PROGRAM Stn10
VAR

	start10: BOOL;
	reset10: BOOL;

	Stn10ProcessFE: F_TRIG;
	Stn10ProcessRE: R_TRIG;
	bCutStn10ProcessHalt: BOOL;
	DoorClose10: R_TRIG;
	bStn10DoorClamp: BOOL;

END_VAR
VAR // added by the converter: edge detectors and wires of the graphical bodies
    _w1, _w2 : ANY;
END_VAR

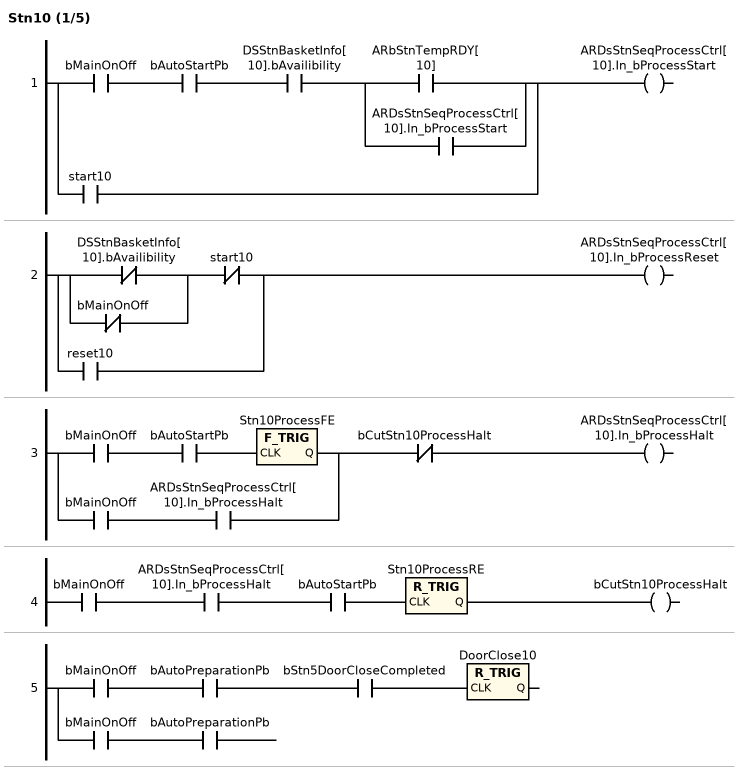
// NETWORK 1
ARDsStnSeqProcessCtrl[10].In_bProcessStart := bMainOnOff AND bAutoStartPb AND DSStnBasketInfo[10].bAvailibility AND (ARbStnTempRDY[10] OR ARDsStnSeqProcessCtrl[10].In_bProcessStart) OR start10;

// NETWORK 2
ARDsStnSeqProcessCtrl[10].In_bProcessReset := (NOT DSStnBasketInfo[10].bAvailibility OR NOT bMainOnOff) AND NOT start10 OR reset10;

// NETWORK 3
Stn10ProcessFE(CLK := bMainOnOff AND bAutoStartPb); // F_TRIG
ARDsStnSeqProcessCtrl[10].In_bProcessHalt := (Stn10ProcessFE.Q OR bMainOnOff AND ARDsStnSeqProcessCtrl[10].In_bProcessHalt) AND NOT bCutStn10ProcessHalt;

// NETWORK 4
Stn10ProcessRE(CLK := bMainOnOff AND ARDsStnSeqProcessCtrl[10].In_bProcessHalt AND bAutoStartPb); // R_TRIG
bCutStn10ProcessHalt := Stn10ProcessRE.Q;

// NETWORK 5
DoorClose10(CLK := bMainOnOff AND bAutoPreparationPb AND bStn5DoorCloseCompleted); // R_TRIG
(* DoorClose10.Q OR bMainOnOff AND bAutoPreparationPb; result not used *)

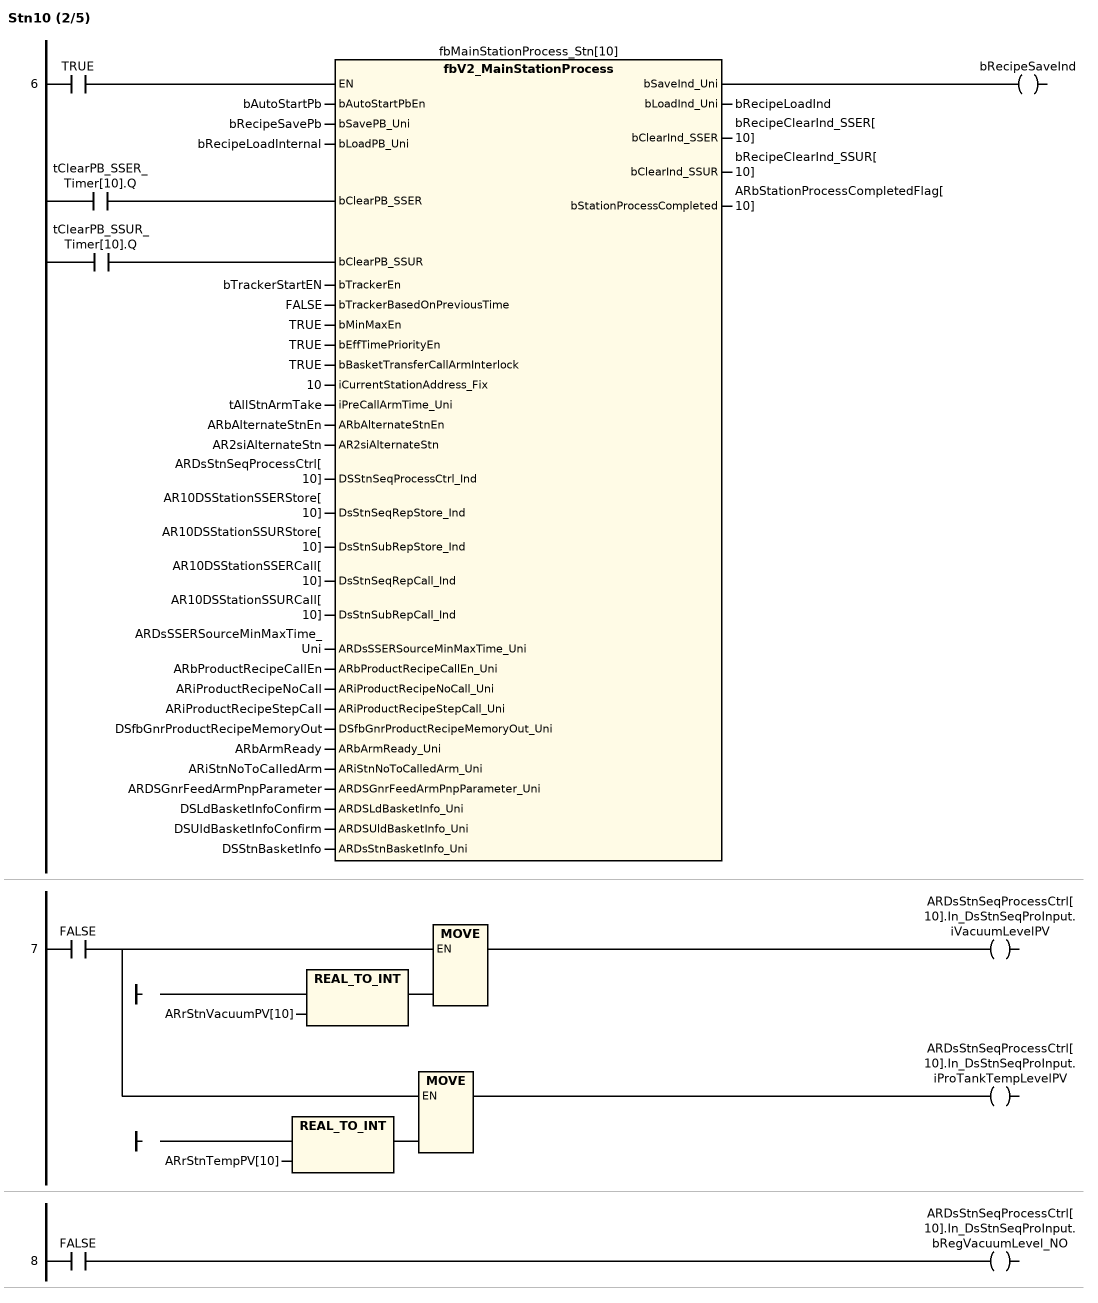
// NETWORK 6
fbMainStationProcess_Stn[10](
    bAutoStartPbEn := bAutoStartPb,
    bSavePB_Uni := bRecipeSavePb,
    bLoadPB_Uni := bRecipeLoadInternal,
    bClearPB_SSER := tClearPB_SSER_Timer[10].Q,
    bClearPB_SSUR := tClearPB_SSUR_Timer[10].Q,
    bTrackerEn := bTrackerStartEN,
    bTrackerBasedOnPreviousTime := FALSE,
    bMinMaxEn := TRUE,
    bEffTimePriorityEn := TRUE,
    bBasketTransferCallArmInterlock := TRUE,
    iCurrentStationAddress_Fix := 10,
    iPreCallArmTime_Uni := tAllStnArmTake,
    ARbAlternateStnEn := ARbAlternateStnEn,
    AR2siAlternateStn := AR2siAlternateStn,
    DSStnSeqProcessCtrl_Ind := ARDsStnSeqProcessCtrl[10],
    DsStnSeqRepStore_Ind := AR10DSStationSSERStore[10],
    DsStnSubRepStore_Ind := AR10DSStationSSURStore[10],
    DsStnSeqRepCall_Ind := AR10DSStationSSERCall[10],
    DsStnSubRepCall_Ind := AR10DSStationSSURCall[10],
    ARDsSSERSourceMinMaxTime_Uni := ARDsSSERSourceMinMaxTime_Uni,
    ARbProductRecipeCallEn_Uni := ARbProductRecipeCallEn,
    ARiProductRecipeNoCall_Uni := ARiProductRecipeNoCall,
    ARiProductRecipeStepCall_Uni := ARiProductRecipeStepCall,
    DSfbGnrProductRecipeMemoryOut_Uni := DSfbGnrProductRecipeMemoryOut,
    ARbArmReady_Uni := ARbArmReady,
    ARiStnNoToCalledArm_Uni := ARiStnNoToCalledArm,
    ARDSGnrFeedArmPnpParameter_Uni := ARDSGnrFeedArmPnpParameter,
    ARDSLdBasketInfo_Uni := DSLdBasketInfoConfirm,
    ARDSUldBasketInfo_Uni := DSUldBasketInfoConfirm,
    ARDsStnBasketInfo_Uni := DSStnBasketInfo,
    bLoadInd_Uni => bRecipeLoadInd,
    bClearInd_SSER => bRecipeClearInd_SSER[10],
    bClearInd_SSUR => bRecipeClearInd_SSUR[10],
    bStationProcessCompleted => ARbStationProcessCompletedFlag[10]); // fbV2_MainStationProcess
bRecipeSaveInd := fbMainStationProcess_Stn[10].bSaveInd_Uni;

// NETWORK 7
IF FALSE THEN _w1 := REAL_TO_INT(ARrStnVacuumPV[10]); END_IF
ARDsStnSeqProcessCtrl[10].In_DsStnSeqProInput.iVacuumLevelPV := _w1;
IF FALSE THEN _w2 := REAL_TO_INT(ARrStnTempPV[10]); END_IF
ARDsStnSeqProcessCtrl[10].In_DsStnSeqProInput.iProTankTempLevelPV := _w2;

// NETWORK 8
ARDsStnSeqProcessCtrl[10].In_DsStnSeqProInput.bRegVacuumLevel_NO := FALSE;

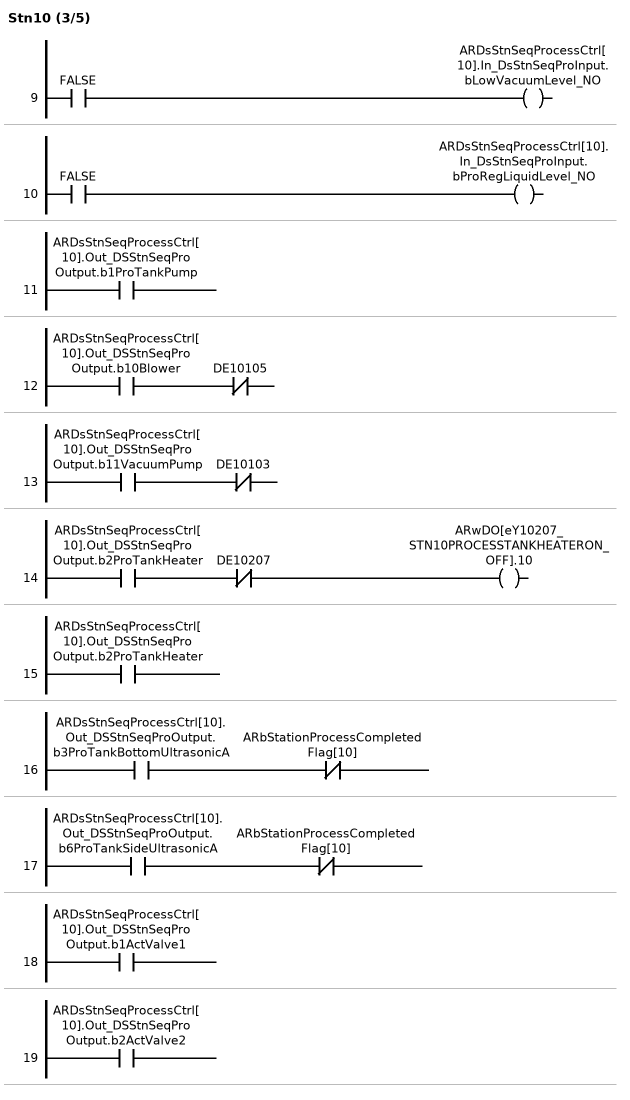
// NETWORK 9
ARDsStnSeqProcessCtrl[10].In_DsStnSeqProInput.bLowVacuumLevel_NO := FALSE;

// NETWORK 10
ARDsStnSeqProcessCtrl[10].In_DsStnSeqProInput.bProRegLiquidLevel_NO := FALSE;

// NETWORK 11
(* ARDsStnSeqProcessCtrl[10].Out_DSStnSeqProOutput.b1ProTankPump; not connected *)

// NETWORK 12
(* ARDsStnSeqProcessCtrl[10].Out_DSStnSeqProOutput.b10Blower AND NOT DE10105; result not used *)

// NETWORK 13
(* ARDsStnSeqProcessCtrl[10].Out_DSStnSeqProOutput.b11VacuumPump AND NOT DE10103; result not used *)

// NETWORK 14
ARwDO[eY10207_STN10PROCESSTANKHEATERON_OFF].10 := ARDsStnSeqProcessCtrl[10].Out_DSStnSeqProOutput.b2ProTankHeater AND NOT DE10207;

// NETWORK 15
(* ARDsStnSeqProcessCtrl[10].Out_DSStnSeqProOutput.b2ProTankHeater; not connected *)

// NETWORK 16
(* ARDsStnSeqProcessCtrl[10].Out_DSStnSeqProOutput.b3ProTankBottomUltrasonicA AND NOT ARbStationProcessCompletedFlag[10]; result not used *)

// NETWORK 17
(* ARDsStnSeqProcessCtrl[10].Out_DSStnSeqProOutput.b6ProTankSideUltrasonicA AND NOT ARbStationProcessCompletedFlag[10]; result not used *)

// NETWORK 18
(* ARDsStnSeqProcessCtrl[10].Out_DSStnSeqProOutput.b1ActValve1; not connected *)

// NETWORK 19
(* ARDsStnSeqProcessCtrl[10].Out_DSStnSeqProOutput.b2ActValve2; not connected *)

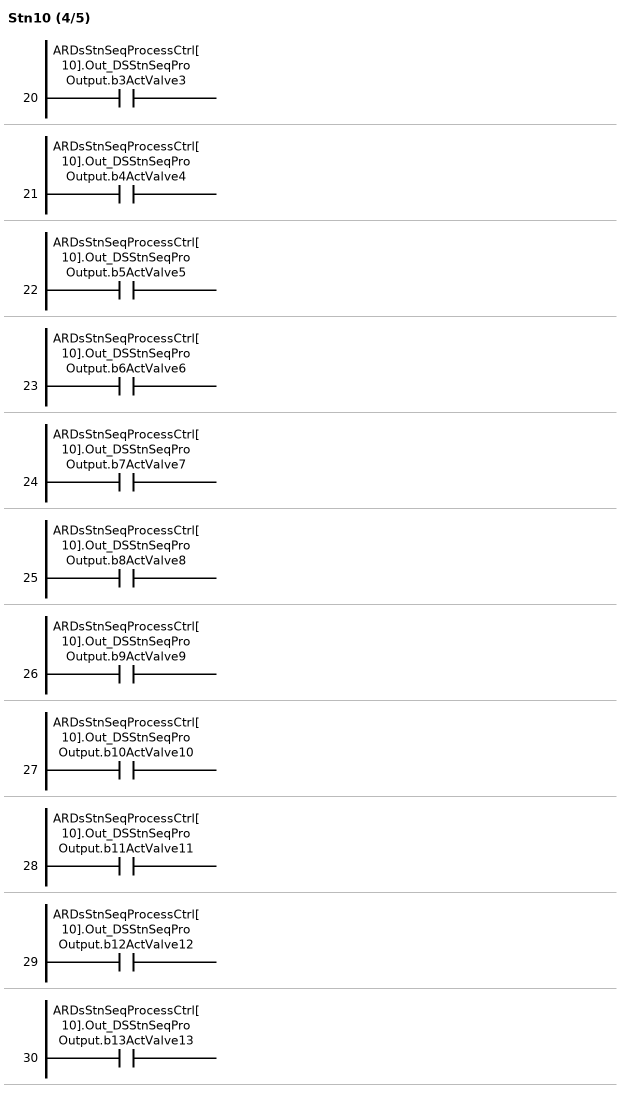
// NETWORK 20
(* ARDsStnSeqProcessCtrl[10].Out_DSStnSeqProOutput.b3ActValve3; not connected *)

// NETWORK 21
(* ARDsStnSeqProcessCtrl[10].Out_DSStnSeqProOutput.b4ActValve4; not connected *)

// NETWORK 22
(* ARDsStnSeqProcessCtrl[10].Out_DSStnSeqProOutput.b5ActValve5; not connected *)

// NETWORK 23
(* ARDsStnSeqProcessCtrl[10].Out_DSStnSeqProOutput.b6ActValve6; not connected *)

// NETWORK 24
(* ARDsStnSeqProcessCtrl[10].Out_DSStnSeqProOutput.b7ActValve7; not connected *)

// NETWORK 25
(* ARDsStnSeqProcessCtrl[10].Out_DSStnSeqProOutput.b8ActValve8; not connected *)

// NETWORK 26
(* ARDsStnSeqProcessCtrl[10].Out_DSStnSeqProOutput.b9ActValve9; not connected *)

// NETWORK 27
(* ARDsStnSeqProcessCtrl[10].Out_DSStnSeqProOutput.b10ActValve10; not connected *)

// NETWORK 28
(* ARDsStnSeqProcessCtrl[10].Out_DSStnSeqProOutput.b11ActValve11; not connected *)

// NETWORK 29
(* ARDsStnSeqProcessCtrl[10].Out_DSStnSeqProOutput.b12ActValve12; not connected *)

// NETWORK 30
(* ARDsStnSeqProcessCtrl[10].Out_DSStnSeqProOutput.b13ActValve13; not connected *)

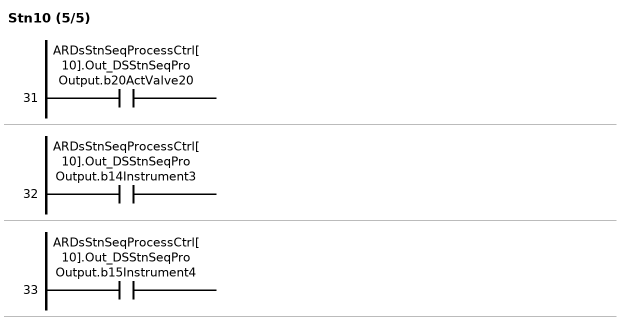
// NETWORK 31
(* ARDsStnSeqProcessCtrl[10].Out_DSStnSeqProOutput.b20ActValve20; not connected *)

// NETWORK 32
(* ARDsStnSeqProcessCtrl[10].Out_DSStnSeqProOutput.b14Instrument3; not connected *)

// NETWORK 33
(* ARDsStnSeqProcessCtrl[10].Out_DSStnSeqProOutput.b15Instrument4; not connected *)

END_PROGRAM

(* stored: Version 1.1.0.1, ProductVersion 3.1.4024.12
   POU Stn10: Id {926dd9c0-77f5-4f96-8875-998085a47073}, SpecialFunc None *)
